FUNCTION_BLOCK FB_VirtualControlBox IMPLEMENTS I_ControlBox
VAR_INPUT
END_VAR
VAR_OUTPUT
END_VAR
VAR
END_VAR

METHOD Joystick
VAR_INPUT
	eMode 	: E_Mode;
	eStatus : E_Status;
END_VAR
VAR_OUTPUT
	fJoystickY : LREAL;
END_VAR
IF eMode = E_Mode.Manual AND eStatus = E_Status.Running THEN
	fJoystickY := G_VirtualControlBox.fJoystickY;
ELSE
	fJoystickY := 0.0;
END_IF
END_METHOD

METHOD Lamps
VAR_INPUT
	eMode 	: E_Mode;
	eStatus : E_Status;
END_VAR
IF eStatus = E_Status.Running AND NOT(eMode = E_Mode.Off) THEN
	G_VirtualControlBox.bGreenLight :=  TRUE;
ELSE
	G_VirtualControlBox.bGreenLight :=  FALSE;
END_IF

IF eStatus = E_Status.Fault  AND NOT(eMode = E_Mode.Off) THEN
	G_VirtualControlBox.bRedLight :=  TRUE;
ELSE
	G_VirtualControlBox.bRedLight :=  FALSE;
END_IF
END_METHOD

METHOD ModeSelector 
VAR_INPUT
END_VAR
VAR_OUTPUT
	eMode : E_Mode;
END_VAR
CASE eMode OF 
	E_Mode.Off:	
		IF G_VirtualControlBox.bOnSelector AND NOT(G_VirtualControlBox.bAutoSelector) THEN	
			eMode := E_Mode.Manual;
		END_IF
		
		IF G_VirtualControlBox.bOnSelector AND G_VirtualControlBox.bAutoSelector THEN	
			eMode := E_Mode.Auto;
		END_IF

	E_Mode.Manual: 
		IF NOT(G_VirtualControlBox.bOnSelector) THEN	
			eMode := E_Mode.Off;
		END_IF
		
		IF G_VirtualControlBox.bOnSelector AND G_VirtualControlBox.bAutoSelector THEN	
			eMode := E_Mode.Auto;
		END_IF
	
	E_Mode.Auto:
		IF NOT(G_VirtualControlBox.bOnSelector) THEN	
			eMode := E_Mode.Off;
		END_IF
		
		IF G_VirtualControlBox.bOnSelector AND NOT(G_VirtualControlBox.bAutoSelector) THEN	
			eMode := E_Mode.Manual;
		END_IF	
ELSE 	
	eMode := E_Mode.Off;
END_CASE
END_METHOD

METHOD PushButtons
VAR_INPUT
	eMode 	: E_Mode;
	eStatus : E_Status;
END_VAR
VAR_OUTPUT
	bStart : BOOL;
	bStop : BOOL;
END_VAR
IF NOT(eMode = E_Mode.Off) AND (NOT(eStatus = E_Status.Fault) OR (eStatus = E_Status.Off)) THEN 
	bStart := G_VirtualControlBox.bStartButton;
	bStop := G_VirtualControlBox.bStopButton;
ELSE
	bStart := FALSE;
	bStop := FALSE;
END_IF
END_METHOD

END_FUNCTION_BLOCK

(* stored: Version 1.1.0.1, ProductVersion 3.1.4024.10
   POU FB_VirtualControlBox: Id {b5dbd877-8357-49f5-a98a-ac539e1b1d21}, SpecialFunc None
   Method Joystick: Id {0e45108c-98eb-4a1c-a573-38934797d553}
   Method Lamps: Id {0dd9b505-9eff-424c-bfde-77014d6169c5}
   Method ModeSelector: Id {e15f3617-ec38-4567-aa4b-7e33c463052d}
   Method PushButtons: Id {eb5d4ee8-8d07-4405-bec2-29949ecb2e14} *)
